# B&R Automation Studio project ui_test
Automation Studio 4.12.2.93; technology packages: mappView 5.19.0

## Configuration TS_UnitTest_Sample

CPU , AutomationRuntime F4.44, Build 6.3.0

### Task classes (Cpu.sw)
```
Cyclic#4 (cycle 10000 us, tolerance 10000000 us):
  SPL_CalcTe <- TS_UnitTest.Samples.Tests_Program.Tests_MyCalcLib_C.SPL_CalcTest.prg
  SPL_CalcT1 <- TS_UnitTest.Samples.Tests_Program.Tests_MyCalcLib_C.SPL_CalcTest_Variants.prg
  SPL_Assert <- TS_UnitTest.Samples.Framework_Extension_With_Custom_Asserts.SPL_AssertsEx.prg
  SPL_Asser1 <- TS_UnitTest.Samples.Framework_Features.SPL_Asserts.prg
  SPL_Behavi <- TS_UnitTest.Samples.Framework_Features.SPL_Behavior.prg
  utTemplate <- TS_UnitTest.Templates.HelperTool_Supported.utTemplate_automated.prg
  utTemplat1 <- TS_UnitTest.Templates.NoToolSupport.utTemplate_manual.prg
Binaries: iomap, asfw, arconfig, ashwd, sysconf
Libraries: Runtime, sys_lib, AsIecCon, astime, AsARCfg, AsBrStr, UnitTest, LibAssert1, UtWs, UtMgr, SPLMyCalc
```

### Hardware
```
PC_any : PC_any v1.1.0.0 (OrderNumber=PC)
  Cyclic1Duration = 100000
  Cyclic1Tolerance = 10000000
  Cyclic2Duration = 200000
  Cyclic2Tolerance = 10000000
  Cyclic3Duration = 500000
  Cyclic3Tolerance = 10000000
  Cyclic4Duration = 10000
  Cyclic4Tolerance = 10000000
  Cyclic5Duration = 2000000
  Cyclic5Tolerance = 10000000
  Cyclic6Duration = 3000000
  Cyclic6Tolerance = 12000000
  Cyclic7Duration = 4000000
  Cyclic7Tolerance = 12000000
  Cyclic8Duration = 5000000
  Cyclic8Tolerance = 30000000
```

## Configuration benchtop

CPU X20CP1381, AutomationRuntime G4.83, Build 4.1.2, Safety 0.0, Vc V4.72.6

### Task classes (Cpu.sw)
```
Cyclic#4:
  Program <- Program.prg
Libraries: AsBrStr, AsARCfg, runtime, sys_lib
```

### Hardware
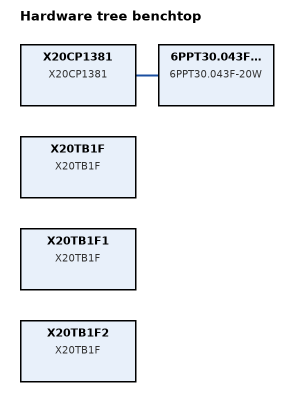
```
6PPT30.043F-20W : 6PPT30.043F-20W v1.3.5.0  [ETH1 -> X20CP1381.IF2 [Cable Type=PowerlinkCable, Length=10, Version=1.0.0.3]]
  Terminal = true
  PasswordVNC = 
  PasswordCIFS = 
  PasswordService = 
  VncKeyMappingFile = VC\6PPT30.043F-20W.dis
X20CP1381 : X20CP1381 v1.14.0.0  [X1 -> X1.SL; X2 -> X2.SL; X3 -> X3.SL]
  Module X1 (Type=X1, Virtual=true, Version=1.14.0.0)
    Connection (Connector=SS1, TargetModule=X20TB1F, TargetConnector=SS)
    Connection (Connector=SL, TargetModule=X20CP1381, TargetConnector=X1)
  Module X2 (Type=X2, Virtual=true, Version=1.14.0.0)
    Connection (Connector=SS1, TargetModule=X20TB1F1, TargetConnector=SS)
    Connection (Connector=SL, TargetModule=X20CP1381, TargetConnector=X2)
  Module X3 (Type=X3, Virtual=true, Version=1.14.0.0)
    Connection (Connector=SS1, TargetModule=X20TB1F2, TargetConnector=SS)
    Connection (Connector=SL, TargetModule=X20CP1381, TargetConnector=X3)
  Connector IF2:
    ActivateDevice = 1
  ConfigurationID = ui_test_benchtop
  ActivateOpcUa = 1
  OpcUaInformationModels_PV_Version = 1
X20TB1F : X20TB1F v1.0.0.0
X20TB1F1 : X20TB1F v1.0.0.0
X20TB1F2 : X20TB1F v1.0.0.0
```

## Logical view

Binary libraries used (declarations not repeated): operator, runtime, astime, AsIecCon, AsBrStr, AsARCfg, sys_lib, UnitTest, UtMgr, UtWs

### Global.var - Global variables
```iecst
VAR
	CurrentTemperature : INT;
	SetTemperature : INT;
END_VAR
```

### Package Logical/Libraries - Global libraries

- Visualisation Logical/mappView (not shown)

### Program Logical/Program (IEC)

#### Main.st
```iecst
PROGRAM _INIT
	SetTemperature := 35;
	CurrentTemperature;

END_PROGRAM

PROGRAM _CYCLIC

END_PROGRAM
```

### Package Logical/TS_UnitTest/Samples/Tests_Program - Unit test sample

### Library Logical/TS_UnitTest/Samples/Tests_Program/SPLMyCalc (IEC) - Simple Calculator
Depends on: Runtime

#### SPLMyCalc.typ - Exported data types
```iecst
(********************************************************************
 * COPYRIGHT -- Bernecker + Rainer
 ********************************************************************
 * Library: SPLMyCalc
 * File: SPLMyCalc.typ
 * Author: B+R
 ********************************************************************
 * Data types of library SPLMyCalc
 ********************************************************************)

TYPE
	MyCalcOperator_enum :
		( (*Enumerator of maths operations*)
		splMyCalcOPERATOR_RESET_OUTPUTS := 0, (*Resets the outputs. No calculation*)
		splMyCalcOPERATOR_ADD := 1, (*Add *)
		splMyCalcOPERATOR_SUBTRACT := 2, (*Subtract*)
		splMyCalcOPERATOR_MULTIPLICATION := 3, (*Multiplication*)
		splMyCalcOPERATOR_DIVISION := 4, (*Division*)
		splMyCalcOPERATOR_SQUARE := 5, (*Square of Param 1*)
		splMyCalcOPERATOR_EXP := 6 (*Param1 ^ Param2*)
		);
END_TYPE
```

#### SPLMyCalc.var - Exported constants
```iecst
(********************************************************************
 * COPYRIGHT --  Bernecker + Rainer
 ********************************************************************
 * Library: SPLMyCalc
 * File: SPLMyCalc.var
 * Author: B+R
 ********************************************************************
 * Constants of library SPLMyCalc
 ********************************************************************)
VAR CONSTANT
	splMyCalcERR_OUT_OF_RANGE : UINT := 50002;
	splMyCalcERR_NO_VALID_PARAM : UINT := 50001;
END_VAR
```

#### SPLMyCalc.fun - Exported functions and function blocks
```iecst
(********************************************************************
 * COPYRIGHT -- Bernecker + Rainer
 ********************************************************************
 * Library: SPLMyCalc
 * File: MyCalc.fun
 * Author: B+R
 ********************************************************************
 * Functions and function blocks of library SPLMyCalc
 ********************************************************************)

FUNCTION_BLOCK MyCalculator (*This functionblock provides several operations. If result is bigger / smaller than MIN or MAX, MIN or MAX are returned.*)
	VAR_INPUT
		CalcOperator : MyCalcOperator_enum; (*Calculation operation*)
		Param1 : INT; (*Paramerter 1*)
		Param2 : INT; (*Paramerter 2*)
	END_VAR
	VAR_OUTPUT
		Status : UINT; (*execution status: ERR_OK, ... *)
		Result : DINT; (*Result of the operation*)
	END_VAR
END_FUNCTION_BLOCK
```

#### SPLMyCalc.st
```iecst
(********************************************************************
 * COPYRIGHT -- Bernecker + Rainer
 ********************************************************************
 * Library: SPLMyCalc
 * File: SPLMyCalc.st
 * Author: B+R
 ********************************************************************
 * Implementation of library SPLMyCalc
 ********************************************************************)

(* This can be used as a sample for  Test Driven Development (TDD)/ Test First Development
Steps (in a nutshell):
    o Define your API (FB, functions, ...)
		 this is already done for the FB MyCalc
	o Create a new test program (by using the template)
	o Write a test case (e.g. Addition) for this FB.
		The tests should describe the expected behavior.
	o Transfer the test program to the target and run the test in the test view
		The test case will fail
	o Implement this FB (Addition), build and transfer, then run the test again
		The test case will pass
	o Write next test (e.g. Subtraction).
	..
	o Write test for MIN / MAX (underflow/overflow)
   	o Run the tests to verify your implementation.

Note:
	The sample test program in SPL_MyCalcLib_C provides some test cases using this FB.

 *)
FUNCTION_BLOCK MyCalculator

	Status := ERR_NOTIMPLEMENTED;

END_FUNCTION_BLOCK
```

### Package Logical/TS_UnitTest/Samples/Tests_Program/Tests_MyCalcLib_C - Tests SPLMyCalc with library "UnitTest"

### Program Logical/TS_UnitTest/Samples/Tests_Program/Tests_MyCalcLib_C/SPL_CalcTest (ANSIC) - Tests SPLMyCalc with library "UnitTest"

#### variables.var - PVs for the program and test suite
```iecst
(********************************************************************
 * COPYRIGHT -- Bernecker + Rainer
 ********************************************************************
 * Program: SPL_CalcTest
 * Author: B+R
 ********************************************************************
 * Local variables of program SPL_CalcTest
 * General variables - do not change
 ********************************************************************)
(*Describe the test*)
VAR
	Testsuite : UtMgrTestSuite := (Name:='SPL_MyCalcTests',Description:='Tests for MyCalc',Type:=utMgrTEST_TYPE_C,MetaInformation:='Some Meta Information can be added here');
END_VAR
(*Variables used in the tests*)
VAR
	instMyCalc : MyCalculator := (0);
END_VAR
```

#### testSuite.c - Handling of program and test suite
```c
/********************************************************************
 * COPYRIGHT -- Bernecker + Rainer
 ********************************************************************
 * Program: SPL_CalcTest
 * Author: B+R
 ********************************************************************
 * Test registration and handshake
 ********************************************************************/

#include <bur/plctypes.h>

#ifdef _DEFAULT_INCLUDES
#include <AsDefault.h>
#endif

#include "UnitTest.h"

void _INIT initTestSuite(void)
{
	utInit(&Testsuite);
}

void _CYCLIC cyclicWithTest(void)
{
	utCyclic(&Testsuite);
}

void _EXIT exitTestSuite(void)
{
	utExit(&Testsuite);
}
```

#### autoGeneratedFile.c - Auto generated code
```c
/*
B+R UnitTest: This is generated code.
Do not edit! Do not move!
Description: UnitTest Testprogramm infrastructure (List of TestSets).
LastUpdated: 2015-04-14 12:04:18Z
By B+R UnitTest Helper Version: 2.0.0.0
*/
#include "UnitTest.h"

UNITTEST_TESTSET_DECLARATION  testSet_MyCalcLib_Addition;
UNITTEST_TESTSET_DECLARATION  testSet_MyCalcLib_Subtraction;
UNITTEST_TESTSET_DECLARATION  testSet_MyCalcLib_Mult_Div;

UNITTEST_TESTSET_FIXTURES(utTestSets)
{
	new_TestSet(testSet_MyCalcLib_Addition),
	new_TestSet(testSet_MyCalcLib_Subtraction),
	new_TestSet(testSet_MyCalcLib_Mult_Div),
};
UNTITTEST_TESTSET_HANDLER();
```

#### testSet_MyCalcLib_Addition.c - Groups test cases for addition
```c
/********************************************************************
 * COPYRIGHT -- Bernecker + Rainer
 ********************************************************************
 * Program: SPL_CalcTest
 * Author: B+R
 ********************************************************************
 * Test set implementation
 ********************************************************************/

#include <bur/plctypes.h>

#ifdef _DEFAULT_INCLUDES
#include <AsDefault.h>
#endif

#include "UnitTest.h"

_TEST test_Add(void)
{
	/* initialize functionblock parameters */
	instMyCalc.CalcOperator = splMyCalcOPERATOR_ADD;
	instMyCalc.Param1   = 1;
	instMyCalc.Param2   = 2;
	/* call synchron functionblock */
	MyCalculator(&instMyCalc);

	/* check result */
	TEST_ASSERT_EQUAL_INT(3, instMyCalc.Result);
	TEST_ASSERT_EQUAL_INT(ERR_OK, instMyCalc.Status);

	/* test is done */
	TEST_DONE;
}

_TEST testResetOutputParam(void)
{

	/* Do any calculation with a result != 0  */
	instMyCalc.CalcOperator = splMyCalcOPERATOR_ADD;
	instMyCalc.Param1   = 1;
	instMyCalc.Param2   = 2;
	/* call synchron functionblock */
	MyCalculator(&instMyCalc);
	/* Please note: the result of the calculation isn't checked as this is not subject of this test case.	 */

	instMyCalc.CalcOperator = splMyCalcOPERATOR_RESET_OUTPUTS;
	/* call synchron functionblock */
	MyCalculator(&instMyCalc);

	/* check result */
	TEST_ASSERT_EQUAL_INT(0, instMyCalc.Result);
	TEST_ASSERT_EQUAL_INT(ERR_OK, instMyCalc.Status);

	/* test is done */
	TEST_DONE;

}

/* This test case shows an example of a test case that can be "false positive".
	As long as MyCalculator() is not implemented, this test passes.
	As long as instMyCalc.Result already is 0 when this test case will be called, it doesn't check wether the FB was called at all.
	--> There are several methods, to verify the FB was called and changed the variables that are used to prove functionality:
	Choose other parameter for an addition with negative values
	Before calling the FB set the output to any other value than the expected result. (e.g. By using _SETUP_TEST() and / or _TEARDOWN_TEST() )
	...

*/
_TEST test_Addition_negValue_badExampleParameter(void)
{
	/* initialize functionblock parameters */
	instMyCalc.CalcOperator = splMyCalcOPERATOR_ADD;
	instMyCalc.Param1   = -1;
	instMyCalc.Param2   = 1;
	/* call synchron functionblock */
	MyCalculator(&instMyCalc);

	/* check result */
	TEST_ASSERT_EQUAL_INT(0, instMyCalc.Result);
	TEST_ASSERT_EQUAL_INT(ERR_OK, instMyCalc.Status);

	/* test is done */
	TEST_DONE;
}

_TEST test_Addition_negValue(void)
{
	/* initialize functionblock parameters */
	instMyCalc.CalcOperator = splMyCalcOPERATOR_ADD;
	instMyCalc.Param1   = -1;
	instMyCalc.Param2   = 3;
	/* call synchron functionblock */
	MyCalculator(&instMyCalc);

	/* check result */
	TEST_ASSERT_EQUAL_INT(2, instMyCalc.Result);
	TEST_ASSERT_EQUAL_INT(ERR_OK, instMyCalc.Status);

	/* test is done */
	TEST_DONE;
}

/*
B+R UnitTest: This is generated code.
Do not edit! Do not move!
Description: UnitTest Testprogramm infrastructure (TestSet).
LastUpdated: 2015-04-14 12:04:18Z
By B+R UnitTest Helper Version: 2.0.0.0
*/
UNITTEST_FIXTURES(fixtures)
{
	new_TestFixture("test_Add", test_Add),
	new_TestFixture("testResetOutputParam", testResetOutputParam),
	new_TestFixture("test_Addition_negValue_badExampleParameter", test_Addition_negValue_badExampleParameter),
	new_TestFixture("test_Addition_negValue", test_Addition_negValue),
};

UNITTEST_CALLER_COMPLETE_EXPLICIT(testSet_MyCalcLib_Addition, "testSet_MyCalcLib_Addition", 0, 0, fixtures, 0, 0, 0);
```

#### testSet_MyCalcLib_Subtraction.c - Groups test cases for substraction
```c
/********************************************************************
 * COPYRIGHT -- Bernecker + Rainer
 ********************************************************************
 * Program: SPL_CalcTest
 * Author: B+R
 ********************************************************************
 * Test set implementation
 ********************************************************************/

#include <bur/plctypes.h>

#ifdef _DEFAULT_INCLUDES
#include <AsDefault.h>
#endif

#include "UnitTest.h"

_TEST test_Subtract(void)
{
	/* initialize functionblock parameters */
	instMyCalc.CalcOperator = splMyCalcOPERATOR_SUBTRACT;
	instMyCalc.Param1   = 4;
	instMyCalc.Param2   = 2;
	/* call synchron functionblock */
	MyCalculator(&instMyCalc);

	/* check result */
	TEST_ASSERT_EQUAL_INT(2, instMyCalc.Result);
	TEST_ASSERT_EQUAL_INT(ERR_OK, instMyCalc.Status);

	/* test is done */
	TEST_DONE;
}

_TEST test_Subtract_negResult(void)
{
	/* initialize functionblock parameters */
	instMyCalc.CalcOperator = splMyCalcOPERATOR_SUBTRACT;
	instMyCalc.Param1   = 6;
	instMyCalc.Param2   = 8;
	/* call synchron functionblock */
	MyCalculator(&instMyCalc);

	/* check result */
	TEST_ASSERT_EQUAL_INT(-2, instMyCalc.Result);
	TEST_ASSERT_EQUAL_INT(ERR_OK, instMyCalc.Status);

	/* test is done */
	TEST_DONE;
}

_TEST test_Subtract_zeroResult(void)
{
	/* initialize functionblock parameters */
	instMyCalc.CalcOperator = splMyCalcOPERATOR_SUBTRACT;
	instMyCalc.Param1   = 6;
	instMyCalc.Param2   = 6;
	/* call synchron functionblock */
	MyCalculator(&instMyCalc);

	/* check result */
	TEST_ASSERT_EQUAL_INT(0, instMyCalc.Result);
	TEST_ASSERT_EQUAL_INT(ERR_OK, instMyCalc.Status);

	/* test is done */
	TEST_DONE;
}

_TEST test_Subtract_boundaryArea_expect_MIN(void)
{
	/* initialize functionblock parameters */
	instMyCalc.CalcOperator = splMyCalcOPERATOR_SUBTRACT;
	instMyCalc.Param1   = -1;
	instMyCalc.Param2   = 32768;
	/* call synchron functionblock */
	MyCalculator(&instMyCalc);

	/* check result */
	TEST_ASSERT_EQUAL_INT(-32768, instMyCalc.Result);
	TEST_ASSERT_EQUAL_INT(splMyCalcERR_OUT_OF_RANGE, instMyCalc.Status);

	/* test is done */
	TEST_DONE;
}

/*
B+R UnitTest: This is generated code.
Do not edit! Do not move!
Description: UnitTest Testprogramm infrastructure (TestSet).
LastUpdated: 2015-04-14 12:04:18Z
By B+R UnitTest Helper Version: 2.0.0.0
*/
UNITTEST_FIXTURES(fixtures)
{
	new_TestFixture("test_Subtract", test_Subtract),
	new_TestFixture("test_Subtract_negResult", test_Subtract_negResult),
	new_TestFixture("test_Subtract_zeroResult", test_Subtract_zeroResult),
	new_TestFixture("test_Subtract_boundaryArea_expect_MIN", test_Subtract_boundaryArea_expect_MIN),
};

UNITTEST_CALLER_COMPLETE_EXPLICIT(testSet_MyCalcLib_Subtraction, "testSet_MyCalcLib_Subtraction", 0, 0, fixtures, 0, 0, 0);
```

#### testSet_MyCalcLib_Mult_Div.c - Groups test cases for multiplication and division
```c
/********************************************************************
 * COPYRIGHT -- Bernecker + Rainer
 ********************************************************************
 * Program: SPL_CalcTest
 * Author: B+R
 ********************************************************************
 * Test set implementation
 ********************************************************************/

#include <bur/plctypes.h>

#ifdef _DEFAULT_INCLUDES
#include <AsDefault.h>
#endif

#include "UnitTest.h"

_TEST test_Multiplication(void)
{
	/* initialize functionblock parameters */
	instMyCalc.CalcOperator = splMyCalcOPERATOR_MULTIPLICATION;
	instMyCalc.Param1   = 4;
	instMyCalc.Param2   = 4;
	/* call synchron functionblock */
	MyCalculator(&instMyCalc);
	/* check result */
	TEST_ASSERT_EQUAL_INT(16, instMyCalc.Result);
	TEST_ASSERT_EQUAL_INT(ERR_OK, instMyCalc.Status);
	/* test is done */
	TEST_DONE;
}

_TEST test_Division(void)
{
	/* initialize functionblock parameters */
	instMyCalc.CalcOperator = splMyCalcOPERATOR_DIVISION;
	instMyCalc.Param1   = 4;
	instMyCalc.Param2   = 4;
	/* call synchron functionblock */
	MyCalculator(&instMyCalc);

	/* check result */
	TEST_ASSERT_EQUAL_INT(1, instMyCalc.Result);
	TEST_ASSERT_EQUAL_INT(ERR_OK, instMyCalc.Status);

	/* test is done */
	TEST_DONE;
}

/*
B+R UnitTest: This is generated code.
Do not edit! Do not move!
Description: UnitTest Testprogramm infrastructure (TestSet).
LastUpdated: 2015-04-14 12:04:18Z
By B+R UnitTest Helper Version: 2.0.0.0
*/
UNITTEST_FIXTURES(fixtures)
{
	new_TestFixture("test_Multiplication", test_Multiplication),
	new_TestFixture("test_Division", test_Division),
};

UNITTEST_CALLER_COMPLETE_EXPLICIT(testSet_MyCalcLib_Mult_Div, "testSet_MyCalcLib_Mult_Div", 0, 0, fixtures, 0, 0, 0);
```

### Program Logical/TS_UnitTest/Samples/Tests_Program/Tests_MyCalcLib_C/SPL_CalcTest_Variants (ANSIC) - Examples how to avoid duplicated test code (advanced)

#### variables.var - PVs for the program and test suite
```iecst
(********************************************************************
 * COPYRIGHT -- Bernecker + Rainer
 ********************************************************************
 * Program: SPL_CalcTest_Variants
 * Author: B+R
 ********************************************************************
 * Local variables of program SPL_CalcTest_Variants
 * General variables - do not change
 ********************************************************************)
(*Describe the test*)
VAR
	Testsuite : UtMgrTestSuite := (Name:='SPL_CalcTest_Variants',Description:='Tests for MyCalc',Type:=utMgrTEST_TYPE_C,MetaInformation:='Some Meta Information can be added here');
END_VAR
(*Variables used in the tests*)
VAR
	instMyCalc : MyCalculator := (0);
END_VAR
```

#### testSuite.c - Handling of program and test suite
```c
/********************************************************************
 * COPYRIGHT -- Bernecker + Rainer
 ********************************************************************
 * Program: SPL_CalcTest_Variants
 * Author: B+R
 ********************************************************************
 * Test registration and handshake
 ********************************************************************/

#include <bur/plctypes.h>

#ifdef _DEFAULT_INCLUDES
#include <AsDefault.h>
#endif

#include "UnitTest.h"

void _INIT initTestSuite(void)
{
	utInit(&Testsuite);
}

void _CYCLIC cyclicWithTest(void)
{
	utCyclic(&Testsuite);
}

void _EXIT exitTestSuite(void)
{
	utExit(&Testsuite);
}
```

#### autoGeneratedFile.c - Auto generated code
```c
/*
B+R UnitTest: This is generated code.
Do not edit! Do not move!
Description: UnitTest Testprogramm infrastructure (List of TestSets).
LastUpdated: 2015-04-14 12:04:18Z
By B+R UnitTest Helper Version: 2.0.0.0
*/
#include "UnitTest.h"

UNITTEST_TESTSET_DECLARATION  testSet_MyCalcLib_Subtraction;
UNITTEST_TESTSET_DECLARATION  testSet_MyCalcLib_Subtraction_variantA;
UNITTEST_TESTSET_DECLARATION  testSet_MyCalcLib_Subtraction_variantB;
UNITTEST_TESTSET_DECLARATION  testSet_MyCalcLib_Subtraction_variantC;
UNITTEST_TESTSET_DECLARATION  testSet_MyCalcLib_Subtraction_variantD;

UNITTEST_TESTSET_FIXTURES(utTestSets)
{
	new_TestSet(testSet_MyCalcLib_Subtraction),
	new_TestSet(testSet_MyCalcLib_Subtraction_variantA),
	new_TestSet(testSet_MyCalcLib_Subtraction_variantB),
	new_TestSet(testSet_MyCalcLib_Subtraction_variantC),
	new_TestSet(testSet_MyCalcLib_Subtraction_variantD),
};
UNTITTEST_TESTSET_HANDLER();
```

#### testSet_MyCalcLib_Subtraction.c - Groups test cases for substraction
```c
/********************************************************************
 * COPYRIGHT -- Bernecker + Rainer
 ********************************************************************
 * Program: SPL_CalcTest_Variants
 * Author: B+R
 ********************************************************************
 * Test set implementation
 ********************************************************************/

#include <bur/plctypes.h>

#ifdef _DEFAULT_INCLUDES
#include <AsDefault.h>
#endif

#include "UnitTest.h"

_TEST test_Subtract(void)
{
	/* initialize functionblock parameters */
	instMyCalc.CalcOperator = splMyCalcOPERATOR_SUBTRACT;
	instMyCalc.Param1   = 4;
	instMyCalc.Param2   = 2;
	/* call synchron functionblock */
	MyCalculator(&instMyCalc);

	/* check result */
	TEST_ASSERT_EQUAL_INT(2, instMyCalc.Result);
	TEST_ASSERT_EQUAL_INT(ERR_OK, instMyCalc.Status);

	/* test is done */
	TEST_DONE;
}

_TEST test_Subtract_negResult(void)
{
	/* initialize functionblock parameters */
	instMyCalc.CalcOperator = splMyCalcOPERATOR_SUBTRACT;
	instMyCalc.Param1   = 6;
	instMyCalc.Param2   = 8;
	/* call synchron functionblock */
	MyCalculator(&instMyCalc);

	/* check result */
	TEST_ASSERT_EQUAL_INT(-2, instMyCalc.Result);
	TEST_ASSERT_EQUAL_INT(ERR_OK, instMyCalc.Status);

	/* test is done */
	TEST_DONE;
}

_TEST test_Subtract_zeroResult(void)
{
	/* initialize functionblock parameters */
	instMyCalc.CalcOperator = splMyCalcOPERATOR_SUBTRACT;
	instMyCalc.Param1   = 6;
	instMyCalc.Param2   = 6;
	/* call synchron functionblock */
	MyCalculator(&instMyCalc);

	/* check result */
	TEST_ASSERT_EQUAL_INT(0, instMyCalc.Result);
	TEST_ASSERT_EQUAL_INT(ERR_OK, instMyCalc.Status);

	/* test is done */
	TEST_DONE;
}

_TEST test_Subtract_boundaryArea_expect_MIN(void)
{
	/* initialize functionblock parameters */
	instMyCalc.CalcOperator = splMyCalcOPERATOR_SUBTRACT;
	instMyCalc.Param1   = -1;
	instMyCalc.Param2   = 32768;
	/* call synchron functionblock */
	MyCalculator(&instMyCalc);

	/* check result */
	TEST_ASSERT_EQUAL_INT(-32768, instMyCalc.Result);
	TEST_ASSERT_EQUAL_INT(splMyCalcERR_OUT_OF_RANGE, instMyCalc.Status);

	/* test is done */
	TEST_DONE;
}

/*
B+R UnitTest: This is generated code.
Do not edit! Do not move!
Description: UnitTest Testprogramm infrastructure (TestSet).
LastUpdated: 2015-04-14 12:04:18Z
By B+R UnitTest Helper Version: 2.0.0.0
*/
UNITTEST_FIXTURES(fixtures)
{
	new_TestFixture("test_Subtract", test_Subtract),
	new_TestFixture("test_Subtract_negResult", test_Subtract_negResult),
	new_TestFixture("test_Subtract_zeroResult", test_Subtract_zeroResult),
	new_TestFixture("test_Subtract_boundaryArea_expect_MIN", test_Subtract_boundaryArea_expect_MIN),
};

UNITTEST_CALLER_COMPLETE_EXPLICIT(testSet_MyCalcLib_Subtraction, "testSet_MyCalcLib_Subtraction", 0, 0, fixtures, 0, 0, 0);
```

#### testSet_MyCalcLib_Subtraction_variantA.c -  To check multiple subtraction combinations without code duplication a helper function can be created.
```c
/********************************************************************
 * COPYRIGHT -- Bernecker + Rainer
 ********************************************************************
 * Program: SPL_CalcTest_Variants
 * Author: B+R
 ********************************************************************
 * Test set implementation
 ********************************************************************/

#include <bur/plctypes.h>

#ifdef _DEFAULT_INCLUDES
#include <AsDefault.h>
#endif

#include "UnitTest.h"

/* To check multiple subtraction combinations without code duplication a helper function can be created.

Note: If an check (assert) is extracted into a helper function, the error report do not contain information about the parameters this helper function was called. For some use cases, this will be acceptable/OK for others not.
	See test_Subtract_MultipleCases()
One option to avoid this is to create multiple Test Cases each calling the same helper function once but with different parameters.
	See test_Subtract_1() and test_Subtract_boundaryArea_expect_MIN()  */
void verify_subtract(INT par1, INT par2 , DINT expectResult)
{
	instMyCalc.CalcOperator = splMyCalcOPERATOR_SUBTRACT;
	instMyCalc.Param1   = par1;
	instMyCalc.Param2   = par2;
	/* call synchron functionblock */
	MyCalculator(&instMyCalc);
	/* check result */
	TEST_ASSERT_EQUAL_INT(expectResult, instMyCalc.Result);
	TEST_ASSERT_EQUAL_INT(ERR_OK, instMyCalc.Status);
}

_TEST test_Subtract(void)
{
	verify_subtract(4, 2,2);

	/* test is done */
	TEST_DONE;
}

_TEST test_Subtract_negResult(void)
{
	verify_subtract(6, 8, -2);

	/* test is done */
	TEST_DONE;
}

_TEST test_Subtract_zeroResult(void)
{
	verify_subtract(6, 6, 0);

	/* test is done */
	TEST_DONE;
}

/* This test isn't reduced as there is (currently) no argument for  instMyCalc.Status  */
_TEST test_Subtract_boundaryArea_expect_MIN(void)
{
	/* initialize functionblock parameters */
	instMyCalc.CalcOperator = splMyCalcOPERATOR_SUBTRACT;
	instMyCalc.Param1   = -1;
	instMyCalc.Param2   = 32768;
	/* call synchron functionblock */
	MyCalculator(&instMyCalc);

	/* check result */
	TEST_ASSERT_EQUAL_INT(-32768, instMyCalc.Result);
	TEST_ASSERT_EQUAL_INT(splMyCalcERR_OUT_OF_RANGE, instMyCalc.Status);

	/* test is done */
	TEST_DONE;
}

/*
B+R UnitTest: This is generated code.
Do not edit! Do not move!
Description: UnitTest Testprogramm infrastructure (TestSet).
LastUpdated: 2015-04-14 12:04:18Z
By B+R UnitTest Helper Version: 2.0.0.0
*/
UNITTEST_FIXTURES(fixtures)
{
	new_TestFixture("test_Subtract", test_Subtract),
	new_TestFixture("test_Subtract_negResult", test_Subtract_negResult),
	new_TestFixture("test_Subtract_zeroResult", test_Subtract_zeroResult),
	new_TestFixture("test_Subtract_boundaryArea_expect_MIN", test_Subtract_boundaryArea_expect_MIN),
};

UNITTEST_CALLER_COMPLETE_EXPLICIT(testSet_MyCalcLib_Subtraction_variantA, "testSet_MyCalcLib_Subtraction_variantA", 0, 0, fixtures, 0, 0, 0);
```

#### testSet_MyCalcLib_Subtraction_variantB.c - TEST_ASSERT is used to output the parameters passed to the helper function when helper returns a failed.
```c
/********************************************************************
 * COPYRIGHT -- Bernecker + Rainer
 ********************************************************************
 * Program: SPL_CalcTest_Variants
 * Author: B+R
 ********************************************************************
 * Test set implementation
 ********************************************************************/

#include <bur/plctypes.h>

#ifdef _DEFAULT_INCLUDES
#include <AsDefault.h>
#endif

#include "UnitTest.h"

/* 	Create a helper returning a BOOL and pass the result of the helper to e.g. TEST_ASSERT()
Note: if the validation itself is not trivial, this function should be tested as well.

If the assert would be used in the helper as well, each of the checks count's twice.
Option would be, to use the TEST_INFO_LOC if returned false. */
BOOL verify_subtract_retBool(INT par1, INT par2 , DINT expectResult)
{
	instMyCalc.CalcOperator = splMyCalcOPERATOR_SUBTRACT;
	instMyCalc.Param1   = par1;
	instMyCalc.Param2   = par2;
	/* call synchron functionblock */
	MyCalculator(&instMyCalc);
	/* check result */
	return (expectResult == instMyCalc.Result);
}

_TEST test_Subtract(void)
{
	TEST_ASSERT(verify_subtract_retBool(4, 2, 2));

	/* test is done */
	TEST_DONE;
}

_TEST test_Subtract_negResult(void)
{
	TEST_ASSERT(verify_subtract_retBool(6, 8, -2));

	/* test is done */
	TEST_DONE;
}

_TEST test_Subtract_zeroResult(void)
{
	TEST_ASSERT(verify_subtract_retBool(6, 6, 0));

	/* test is done */
	TEST_DONE;
}

/* This test isn't reduced as there is (currently) no argument for  instMyCalc.Status  */
_TEST test_Subtract_boundaryArea_expect_MIN(void)
{
	/* initialize functionblock parameters */
	instMyCalc.CalcOperator = splMyCalcOPERATOR_SUBTRACT;
	instMyCalc.Param1   = -1;
	instMyCalc.Param2   = 32768;
	/* call synchron functionblock */
	MyCalculator(&instMyCalc);

	/* check result */
	TEST_ASSERT_EQUAL_INT(-32768, instMyCalc.Result);
	TEST_ASSERT_EQUAL_INT(splMyCalcERR_OUT_OF_RANGE, instMyCalc.Status);

	/* test is done */
	TEST_DONE;
}

/*
B+R UnitTest: This is generated code.
Do not edit! Do not move!
Description: UnitTest Testprogramm infrastructure (TestSet).
LastUpdated: 2015-04-14 12:04:18Z
By B+R UnitTest Helper Version: 2.0.0.0
*/
UNITTEST_FIXTURES(fixtures)
{
	new_TestFixture("test_Subtract", test_Subtract),
	new_TestFixture("test_Subtract_negResult", test_Subtract_negResult),
	new_TestFixture("test_Subtract_zeroResult", test_Subtract_zeroResult),
	new_TestFixture("test_Subtract_boundaryArea_expect_MIN", test_Subtract_boundaryArea_expect_MIN),
};

UNITTEST_CALLER_COMPLETE_EXPLICIT(testSet_MyCalcLib_Subtraction_variantB, "testSet_MyCalcLib_Subtraction_variantB", 0, 0, fixtures, 0, 0, 0);
```

#### testSet_MyCalcLib_Subtraction_variantC.c - When the helper is formulated as macro, the correct location (line / file) inside the testcase is given.
```c
/********************************************************************
 * COPYRIGHT -- Bernecker + Rainer
 ********************************************************************
 * Program: SPL_CalcTest_Variants
 * Author: B+R
 ********************************************************************
 * Test set implementation
 ********************************************************************/

#include <bur/plctypes.h>

#ifdef _DEFAULT_INCLUDES
#include <AsDefault.h>
#endif

#include "UnitTest.h"

#ifdef SMARTEDIT_DUMMY
/* When the helper is formulated as macro, the correct location (line / file) inside the testcase is given.
Each time the macro is used, the code gets duplicated.

Best practise: Extract a helper function first, use / test it before converting it into a macro, as functions can be far farbetter debugged / analyzed than macros. */
void def_verify_subtract(INT par1, INT par2 , DINT expectResult);
#endif
#define  def_verify_subtract( par1,  par2 , expectResult)\
{\
	instMyCalc.CalcOperator = splMyCalcOPERATOR_SUBTRACT;\
	instMyCalc.Param1   = par1;\
	instMyCalc.Param2   = par2;\
	/* call synchron functionblock */\
	MyCalculator(&instMyCalc);\
	/* check result */\
	TEST_ASSERT_EQUAL_INT(expectResult, instMyCalc.Result);\
	TEST_ASSERT_EQUAL_INT(ERR_OK, instMyCalc.Status);\
}

_TEST test_Subtract(void)
{
	def_verify_subtract(4, 2, 2);

	/* test is done */
	TEST_DONE;
}

_TEST test_Subtract_negResult(void)
{
	def_verify_subtract(6, 8, -2);
	/* test is done */
	TEST_DONE;
}

_TEST test_Subtract_zeroResult(void)
{
	def_verify_subtract(6, 6, 0);

	/* test is done */
	TEST_DONE;
}

/* This test isn't reduced as there is (currently) no argument for  instMyCalc.Status  */
_TEST test_Subtract_boundaryArea_expect_MIN(void)
{
	/* initialize functionblock parameters */
	instMyCalc.CalcOperator = splMyCalcOPERATOR_SUBTRACT;
	instMyCalc.Param1   = -1;
	instMyCalc.Param2   = 32768;
	/* call synchron functionblock */
	MyCalculator(&instMyCalc);

	/* check result */
	TEST_ASSERT_EQUAL_INT(-32768, instMyCalc.Result);
	TEST_ASSERT_EQUAL_INT(splMyCalcERR_OUT_OF_RANGE, instMyCalc.Status);

	/* test is done */
	TEST_DONE;
}

/*
B+R UnitTest: This is generated code.
Do not edit! Do not move!
Description: UnitTest Testprogramm infrastructure (TestSet).
LastUpdated: 2015-04-14 12:04:18Z
By B+R UnitTest Helper Version: 2.0.0.0
*/
UNITTEST_FIXTURES(fixtures)
{
	new_TestFixture("test_Subtract", test_Subtract),
	new_TestFixture("test_Subtract_negResult", test_Subtract_negResult),
	new_TestFixture("test_Subtract_zeroResult", test_Subtract_zeroResult),
	new_TestFixture("test_Subtract_boundaryArea_expect_MIN", test_Subtract_boundaryArea_expect_MIN),
};

UNITTEST_CALLER_COMPLETE_EXPLICIT(testSet_MyCalcLib_Subtraction_variantC, "testSet_MyCalcLib_Subtraction_variantC", 0, 0, fixtures, 0, 0, 0);
```

#### testSet_MyCalcLib_Subtraction_variantD.c - Custom Assert
```c
/********************************************************************
 * COPYRIGHT -- Bernecker + Rainer
 ********************************************************************
 * Program: SPL_CalcTest_Variants
 * Author: B+R
 ********************************************************************
 * Test set implementation
 ********************************************************************/

#include <bur/plctypes.h>

#ifdef _DEFAULT_INCLUDES
#include <AsDefault.h>
#endif

#include "UnitTest.h"

/*****************************************
* Begin Custom Assert

* Note: Custom asserts may be seperated from Test Sets.
* 		In this sample it's part of the Test Set file for symmetry reason
*
* Note: To learn more about Custom Asserts see help
*		or sample in \Logical\TS_UnitTest\Samples\Samples_Advanced_CustomAsserts\
 */
BOOL spl_verify_subtract_impl(INT par1, INT par2 , DINT expectResult,  unsigned long line, const char *file)
{
	instMyCalc.CalcOperator = splMyCalcOPERATOR_SUBTRACT;
	instMyCalc.Param1   = par1;
	instMyCalc.Param2   = par2;

	/* call synchron functionblock */
	MyCalculator(&instMyCalc);

	/* check expectations and report outcome */
	if(expectResult != instMyCalc.Result)
	{
		addFailure("Calculation Error", line, file);
	}
	else if (ERR_OK != instMyCalc.Status)
	{
		addFailure("Unexpected Status", line, file);
	}
	else
	{
		addPassed("",0,0);
		return 1;
	}
	return 0;
}

#ifdef SMARTEDIT_DUMMY
/* When the helper is formulated as macro, the correct location (line / file) inside the testcase is given. */
void SPL_ASSERT_VERIFY_SUBTRACT(INT par1, INT par2 , DINT expectResult);
#endif
#define  SPL_ASSERT_VERIFY_SUBTRACT( par1,  par2 , expectResult)  spl_verify_subtract_impl(par1, par2, expectResult, __LINE__, __FILE__);

/*****************************************
* End Custom Assert
*/

/*****************************************
	Begin Test Set
*/
_TEST test_Subtract(void)
{
	SPL_ASSERT_VERIFY_SUBTRACT(4, 2, 2);

	/* test is done */
	TEST_DONE;
}

_TEST test_Subtract_negResult(void)
{
	SPL_ASSERT_VERIFY_SUBTRACT(6, 8, -2);
	/* test is done */
	TEST_DONE;
}

_TEST test_Subtract_zeroResult(void)
{
	SPL_ASSERT_VERIFY_SUBTRACT(6, 6, 0);

	/* test is done */
	TEST_DONE;
}

/* This test isn't reduced as there is (currently) no argument for  instMyCalc.Status  */
_TEST test_Subtract_boundaryArea_expect_MIN(void)
{
	/* initialize functionblock parameters */
	instMyCalc.CalcOperator = splMyCalcOPERATOR_SUBTRACT;
	instMyCalc.Param1   = -1;
	instMyCalc.Param2   = 32768;
	/* call synchron functionblock */
	MyCalculator(&instMyCalc);

	/* check result */
	TEST_ASSERT_EQUAL_INT(-32768, instMyCalc.Result);
	TEST_ASSERT_EQUAL_INT(splMyCalcERR_OUT_OF_RANGE, instMyCalc.Status);

	/* test is done */
	TEST_DONE;
}

/*
B+R UnitTest: This is generated code.
Do not edit! Do not move!
Description: UnitTest Testprogramm infrastructure (TestSet).
LastUpdated: 2015-04-14 12:04:18Z
By B+R UnitTest Helper Version: 2.0.0.0
*/
UNITTEST_FIXTURES(fixtures)
{
	new_TestFixture("test_Subtract", test_Subtract),
	new_TestFixture("test_Subtract_negResult", test_Subtract_negResult),
	new_TestFixture("test_Subtract_zeroResult", test_Subtract_zeroResult),
	new_TestFixture("test_Subtract_boundaryArea_expect_MIN", test_Subtract_boundaryArea_expect_MIN),
};

UNITTEST_CALLER_COMPLETE_EXPLICIT(testSet_MyCalcLib_Subtraction_variantD, "testSet_MyCalcLib_Subtraction_variantD", 0, 0, fixtures, 0, 0, 0);
```

### Package Logical/TS_UnitTest/Samples/Framework_Extension_With_Custom_Asserts - Custom asserts

- Library Logical/TS_UnitTest/Samples/Framework_Extension_With_Custom_Asserts/LibAssert1 (ANSIC) - Sample library: Creation of custom asserts (no source held here)

### Program Logical/TS_UnitTest/Samples/Framework_Extension_With_Custom_Asserts/SPL_AssertsEx (ANSIC) - This sample uses custom asserts defined in LibAssert1

#### README.txt
```
Please note

The samples in this program provides no good programming style!
They are solely for demonstrating the behavior of the framework.
Bad style:
	o	There is no test of any function or FB, just asserts failing or passing (depending on PV values)
	o	Expectations are variables and no constants
	o	Results are constants instead of results / outputs
	o	Mulitple asserts per Test Case
```

#### testSuite.var
```iecst
(********************************************************************
 * COPYRIGHT -- Bernecker + Rainer
 ********************************************************************
 * Program: SPL_AssertsEx
 * Author: B+R
 ********************************************************************
 * Local variables of program SPL_AssertsEx
 * General variables
 ********************************************************************)
VAR
	Testsuite : UtMgrTestSuite := (Name:='SPL_CustomAsserts',Description:='The sample custom asserts are defined in LibAssert1. This test shows their usage.',Type:=utMgrTEST_TYPE_C);
END_VAR
```

#### testSuite.c
```c
/********************************************************************
 * COPYRIGHT -- Bernecker + Rainer
 ********************************************************************
 * Program: SPL_AssertsEx
 * Author: B+R
 ********************************************************************
 * Test registration and handshake
 ********************************************************************/

#include <bur/plctypes.h>

#ifdef _DEFAULT_INCLUDES
#include <AsDefault.h>
#endif

#include "UnitTest.h"

void _INIT initTestSuite(void)
{
	utInit(&Testsuite);
}

void _CYCLIC cyclicWithTest(void)
{
	/* Some code */
	utCyclic(&Testsuite);
}

void _EXIT exitTestSuite(void)
{
	utExit(&Testsuite);
}
```

#### autoGeneratedFile.c
```c
/*
B+R UnitTest: This is generated code.
Do not edit! Do not move!
Description: UnitTest Testprogramm infrastructure (List of TestSets).
LastUpdated: 2015-04-14 12:04:08Z
By B+R UnitTest Helper Version: 2.0.0.0
*/
#include "UnitTest.h"

UNITTEST_TESTSET_DECLARATION  testSet_AssertsExt;

UNITTEST_TESTSET_FIXTURES(utTestSets)
{
	new_TestSet(testSet_AssertsExt),
};
UNTITTEST_TESTSET_HANDLER();
```

#### varAssertExt.var - Variables used in testSet_AssertsExt
```iecst
(********************************************************************
 * COPYRIGHT -- Bernecker + Rainer
 ********************************************************************
 * Program: SPL_AssertsEx
 * Author: B+R
 ********************************************************************
 * Local variables of program SPL_AssertsEx
 * For test set testSet_AssertsExt.c
 ********************************************************************)
VAR
	FloatArrayDeltaForComparison : ARRAY[0..50] OF REAL;
	FloatArray2 : ARRAY[0..50] OF REAL;
	FloatArray1 : ARRAY[0..50] OF REAL;
END_VAR
```

#### testSet_AssertsExt.c - Uses Assertions of Library utAssertExt
```c
/********************************************************************
* COPYRIGHT -- Bernecker + Rainer
********************************************************************
* Program: SPL_AssertsEx
* Author: B+R
********************************************************************
* This test set shows the use of self created asserts.
* Asserts are implemented in the library LibAssert1.
********************************************************************/

#include <bur/plctypes.h>

#ifdef _DEFAULT_INCLUDES
#include <AsDefault.h>
#endif

#include "UnitTest.h"
#include "LibAssert1.h"

_TEST test_splAssert_ArrayOfRealValues(void)
{
	/* manual generated differences for demonstration of the SPL_ASSERT */
	FloatArray1[0] = 2;
	FloatArray2[0] = 2;

	FloatArray1[1] = 3;
	FloatArray2[1] = 1;

	FloatArray1[30] = 3.33;
	FloatArray2[30] = 1.11;

	FloatArrayDeltaForComparison[31] = 1; /* Within -> pass, equal -> failed */
	FloatArray1[31] = 3.33;
	FloatArray2[31] = 3.31;

	SPL_ASSERT_ARRAY_EQUAL_REAL(FloatArray1, FloatArray2, sizeof(FloatArray1) / sizeof(FloatArray1[0]) );
	SPL_ASSERT_ARRAY_REAL_WITHIN(FloatArrayDeltaForComparison, FloatArray1, FloatArray2, sizeof(FloatArray1) / sizeof(FloatArray1[0]) );
	TEST_DONE;
}

_TEST test_splAssert_Boundary()
{
	/* should fail */
	SPL_ASSERT_UPPER_BOUNDARY(2,4);

	/* should pass */
	SPL_ASSERT_UPPER_BOUNDARY(4,2);

	TEST_DONE;
}

/*
B+R UnitTest: This is generated code.
Do not edit! Do not move!
Description: UnitTest Testprogramm infrastructure (TestSet).
LastUpdated: 2015-04-14 12:04:07Z
By B+R UnitTest Helper Version: 2.0.0.0
*/
UNITTEST_FIXTURES(fixtures)
{
	new_TestFixture("test_splAssert_ArrayOfRealValues", test_splAssert_ArrayOfRealValues),
	new_TestFixture("test_splAssert_Boundary", test_splAssert_Boundary),
};

UNITTEST_CALLER_COMPLETE_EXPLICIT(testSet_AssertsExt, "testSet_AssertsExt", 0, 0, fixtures, 0, 0, 0);
```

### Package Logical/TS_UnitTest/Samples/Framework_Features - Framework features

### Program Logical/TS_UnitTest/Samples/Framework_Features/SPL_Asserts (ANSIC) - Available basic asserts

#### README.txt
```
Please note

The samples in this program provides no good programming style!
They are solely for demonstrating the behavior of the framework.
Bad style:
	o	There is no test of any function or FB, just asserts failing or passing (depending on PV values)
	o	Expectations are variables and no constants
	o	Mulitple asserts per Test Case
```

#### testSuite.var
```iecst
(********************************************************************
 * COPYRIGHT -- Bernecker + Rainer
 ********************************************************************
 * Program: SPL_Asserts
 * Author: B+R
 ********************************************************************
 * Local variables of program SPL_Asserts
 * General variables
 ********************************************************************)
VAR
	Testsuite : UtMgrTestSuite := (Name:='SPL_Asserts',Description:='Shows asserts and usage',Type:=utMgrTEST_TYPE_C);
END_VAR
```

#### testSuite.c - Handling of program and test suite
```c
/********************************************************************
 * COPYRIGHT -- Bernecker + Rainer
 ********************************************************************
 * Program: SPL_Asserts
 * Author: B+R
 ********************************************************************
 * Test registration and handshake
 ********************************************************************/

#include <bur/plctypes.h>

#ifdef _DEFAULT_INCLUDES
#include <AsDefault.h>
#endif

#include "UnitTest.h"

void _INIT initTestSuite(void)
{
	utInit(&Testsuite);
}

void _CYCLIC cyclicWithTest(void)
{
	/* Some code */
	utCyclic(&Testsuite);
}

void _EXIT exitTestSuite(void)
{
	utExit(&Testsuite);
}
```

#### autoGeneratedFile.c - Auto generated code
```c
/*
B+R UnitTest: This is generated code.
Do not edit! Do not move!
Description: UnitTest Testprogramm infrastructure (List of TestSets).
LastUpdated: 2015-04-14 12:03:48Z
By B+R UnitTest Helper Version: 2.0.0.0
*/
#include "UnitTest.h"

UNITTEST_TESTSET_DECLARATION  testSet_Asserts;

UNITTEST_TESTSET_FIXTURES(utTestSets)
{
	new_TestSet(testSet_Asserts),
};
UNTITTEST_TESTSET_HANDLER();
```

#### varAsserts.var - Variables used in testSet_Asserts
```iecst
(********************************************************************
 * COPYRIGHT -- Bernecker + Rainer
 ********************************************************************
 * Program: SPL_Asserts
 * Author: B+R
 ********************************************************************
 * Local variables of program SPL_Asserts
 * For test set testSet_Asserts.c
 ********************************************************************)
VAR
	Buffer1 : ARRAY[0..9] OF USINT := [10(0)];
	Buffer2 : ARRAY[0..19] OF USINT := [20(0)];
	MySecondVar : UDINT := 2;
	Pointer : REFERENCE TO UDINT;
	ConditionFlag : BOOL := FALSE;
END_VAR
(*Strings*)
VAR
	String1 : STRING[80] := '';
	String2 : STRING[80] := '';
	WString1 : WSTRING[80] := "World";
	WString2 : WSTRING[80] := "Hello";
END_VAR
(*Integer*)
VAR
	Si1 : SINT := 0;
	Si2 : SINT := 0;
	Usi1 : USINT := 0;
	Usi2 : USINT := 0;
	I1 : INT := 0;
	I2 : INT := 0;
	Ui1 : UINT := 0;
	Ui2 : UINT := 0;
	Di1 : DINT := 0;
	Di2 : DINT := 0;
	Udi1 : UDINT := 0;
	Udi2 : UDINT := 0;
END_VAR
(*Floatingpoint*)
VAR
	LReal2 : REAL;
	LRealDeltaForComparison : REAL;
	LReal1 : REAL;
	Real2 : REAL;
	RealDeltaForComparison : REAL;
	Real1 : REAL;
END_VAR
```

#### testSet_Asserts.c - Available Asserts
```c
/********************************************************************
* COPYRIGHT -- Bernecker + Rainer
********************************************************************
* Program: SPL_Asserts
* Author: B+R
********************************************************************
* This test set shows the available asserts of the UnitTest library
********************************************************************/

#include <bur/plctypes.h>

#ifdef _DEFAULT_INCLUDES
#include <AsDefault.h>
#endif

#include "UnitTest.h"

/* Executed before each test case */
_SETUP_TEST(void)
{
	MySecondVar = 2;

	TEST_DONE;
}

/* Executed after each test case */
_TEARDOWN_TEST(void)
{
	TEST_DONE;
}

_TEST test_int(void)
{
	TEST_ASSERT_EQUAL_INT(	Usi1, 	Usi2);
	TEST_ASSERT_EQUAL_INT( 	Si1,	Si2 );
	TEST_ASSERT_EQUAL_INT( 	Ui1, 	Ui2	);
	TEST_ASSERT_EQUAL_INT( 	I1, 	I2	);
	TEST_ASSERT_EQUAL_INT( 	Di1, 	Di2	);
	TEST_ASSERT_EQUAL_INT(	Udi1, 	Udi2);

	TEST_DONE;
}

_TEST test_string(void)
{
	TEST_ASSERT_EQUAL_STRING(String1, String2 );

	TEST_DONE;
}

_TEST test_wstring(void)
{
	TEST_ASSERT_EQUAL_WSTRING(WString1,	WString2);

	TEST_DONE;
}

_TEST test_float(void)
{
	TEST_ASSERT_EQUAL_FLOAT(Real1, Real2);
	TEST_ASSERT_FLOAT_WITHIN(RealDeltaForComparison, Real1, Real2);

	TEST_ASSERT_EQUAL_REAL(Real1, Real2);
	TEST_ASSERT_REAL_WITHIN(RealDeltaForComparison, Real1, Real2);

	TEST_DONE;
}

_TEST test_double(void)
{
	TEST_ASSERT_EQUAL_DOUBLE(LReal1, LReal2);
	TEST_ASSERT_DOUBLE_WITHIN(LRealDeltaForComparison, LReal1, LReal2);

	TEST_ASSERT_EQUAL_LREAL(LReal1, LReal2);
	TEST_ASSERT_LREAL_WITHIN(LRealDeltaForComparison, LReal1, LReal2);

	TEST_DONE;
}

_TEST test_memory(void)
{
	TEST_ASSERT_EQUAL_MEM(Buffer1, Buffer2, sizeof(Buffer1)  );

	TEST_DONE;
}

_TEST test_null_true_and_false(void)
{
	TEST_ASSERT_NOT_NULL(Pointer);
	TEST_ASSERT_NOT_NULL(0); 	/* Not Ok */

	TEST_ASSERT_NULL(0); 		/* Ok */
	TEST_ASSERT_NULL(Pointer);

	Pointer = &Udi1;
	TEST_ASSERT_NULL(Pointer); /* Not Ok */

	TEST_DONE;
}

_TEST test_message(void)
{
	TEST_ASSERT_MESSAGE(ConditionFlag, "This text, if condition evaluates to false.");
	ConditionFlag = 0;
	TEST_ASSERT_MESSAGE(ConditionFlag, "This text, because condition evaluates to false.");
	ConditionFlag = 4;
	TEST_ASSERT_MESSAGE(ConditionFlag, "Nothing, as condition evaluates to true (!= 0).");

	TEST_DONE;
}

_TEST test_info(void)
{
	TEST_INFO("Info Text - for some comment");
	TEST_INFO_POS("Info Text - for some comment with position");

	TEST_DONE;
}

_TEST test_fail(void)
{
	TEST_FAIL("Always fails");

	TEST_DONE;
}

/*
B+R UnitTest: This is generated code.
Do not edit! Do not move!
Description: UnitTest Testprogramm infrastructure (TestSet).
LastUpdated: 2015-04-14 12:03:48Z
By B+R UnitTest Helper Version: 2.0.0.0
*/
UNITTEST_FIXTURES(fixtures)
{
	new_TestFixture("test_int", test_int),
	new_TestFixture("test_string", test_string),
	new_TestFixture("test_wstring", test_wstring),
	new_TestFixture("test_float", test_float),
	new_TestFixture("test_double", test_double),
	new_TestFixture("test_memory", test_memory),
	new_TestFixture("test_null_true_and_false", test_null_true_and_false),
	new_TestFixture("test_message", test_message),
	new_TestFixture("test_info", test_info),
	new_TestFixture("test_fail", test_fail),
};

UNITTEST_CALLER_COMPLETE_EXPLICIT(testSet_Asserts, "testSet_Asserts", setupTest, teardownTest, fixtures, 0, 0, 0);
```

### Program Logical/TS_UnitTest/Samples/Framework_Features/SPL_Behavior (ANSIC) - This sample is about the control flow of test programs

#### README.txt
```
Please note

The samples in this program provides no good programming style!
They are solely for demonstrating the behavior of the framework.
Bad style:
	o	Asserts should only be used to verify the test case as the report should be short ans meaningful (No explainings, just the relevant facts).
	o	Asserts should only be used in test cases.
	o	Test cases should be named meaningful.
	o	Macros are used instead of helper functions.
```

#### testSuite.var
```iecst
(********************************************************************
 * COPYRIGHT -- Bernecker + Rainer
 ********************************************************************
 * Program: SPL_Behavior
 * Author: B+R
 ********************************************************************
 * Local variables of program SPL_Behavior
 * General variables
 ********************************************************************)
VAR
	Testsuite : UtMgrTestSuite := (Name:='SPL_framework_behavior',Description:='Every TestSet provides an independend sample to show the behavior of a set',Type:=utMgrTEST_TYPE_C);
END_VAR
```

#### testSuite.c - Handling of program and test suite
```c
/********************************************************************
 * COPYRIGHT -- Bernecker + Rainer
 ********************************************************************
 * Program: SPL_Behavior
 * Author: B+R
 ********************************************************************
 * Test registration and handshake
 ********************************************************************/

#include <bur/plctypes.h>

#ifdef _DEFAULT_INCLUDES
#include <AsDefault.h>
#endif

#include "UnitTest.h"

#include "iPrototypes.h"

void _INIT initTestSuite(void)
{
	utInit(&Testsuite);
}

void _CYCLIC cyclicWithTest(void)
{
	/* Some code */
	utCyclic(&Testsuite);

	if(Testsuite.TestFinishedDone)
	{
		resetDataForTestSet_Complete();
		resetDataForTestSet_TestCases();
		resetDataForTestSet_SetSetupTeardown();
		resetDataForTestSet_TestSetupTeardown();
	}
}

void _EXIT exitTestSuite(void)
{
	utExit(&Testsuite);
}
```

#### autoGeneratedFile.c - Auto generated code
```c
/*
B+R UnitTest: This is generated code.
Do not edit! Do not move!
Description: UnitTest Testprogramm infrastructure (List of TestSets).
LastUpdated: 2015-04-14 12:03:48Z
By B+R UnitTest Helper Version: 2.0.0.0
*/
#include "UnitTest.h"

UNITTEST_TESTSET_DECLARATION  test_SetTestCases;
UNITTEST_TESTSET_DECLARATION  test_SetTestCases_SetSetup_SetTeardown;
UNITTEST_TESTSET_DECLARATION  test_SetTestCases_TestSetup_TestTeardown;
UNITTEST_TESTSET_DECLARATION  test_SetComplete;
UNITTEST_TESTSET_DECLARATION  TestBusy_Asyncronous;
UNITTEST_TESTSET_DECLARATION  TestBusy_Asyncronous_with_CyclicSet;

UNITTEST_TESTSET_FIXTURES(utTestSets)
{
	new_TestSet(test_SetTestCases),
	new_TestSet(test_SetTestCases_SetSetup_SetTeardown),
	new_TestSet(test_SetTestCases_TestSetup_TestTeardown),
	new_TestSet(test_SetComplete),
	new_TestSet(TestBusy_Asyncronous),
	new_TestSet(TestBusy_Asyncronous_with_CyclicSet),
};
UNTITTEST_TESTSET_HANDLER();
```

#### iPrototypes.h
```c
/********************************************************************
 * COPYRIGHT -- Bernecker + Rainer
 ********************************************************************
 * Program: SPL_Behavior
 * File: iPrototypes.h
 * Author: B+R
 *******************************************************************/

#include <bur/plctypes.h>

/* Prototyping of functions  */
void 	resetDataForTestSet();
void 	checkAndWriteCounterIfChanged( unsigned long line, const char *file);

void	resetDataForTestSet_Complete();
void	resetDataForTestSet_TestCases();
void	resetDataForTestSet_SetSetupTeardown();
void	resetDataForTestSet_TestSetupTeardown();
```

#### iHelperFunction.h
```c
/********************************************************************
 * COPYRIGHT -- Bernecker + Rainer
 ********************************************************************
 * Program: SPL_Behavior
 * File: iHelperFunction.h
 * Author: B+R
 *******************************************************************/

#include <bur/plctypes.h>

#include "iPrototypes.h"

/* This Macro is for tracing the calls in the sample
(For exemplification)*/
#define LOG_FOR_EXEMPLIFICATION_CYCLIC_SET  \
	brsstrcat((UDINT)OutputString, (UDINT)"Cyclic set - "); \
	checkAndWriteCounterIfChanged(__LINE__, __FILE__); \
	CounterInSet++;

/* This Macro is for tracing the calls in the sample
(For exemplification)*/
#define LOG_FOR_EXEMPLIFICATION_TEST_CASE_1   \
	brsstrcat((UDINT)OutputString,(UDINT) "Call test 1 - "); \
	checkAndWriteCounterIfChanged(__LINE__, __FILE__);

/* This Macro is for tracing the calls in the sample
(For exemplification)*/
#define LOG_FOR_EXEMPLIFICATION_TEST_CASE_2 \
	brsstrcat((UDINT)OutputString,(UDINT) "Call test 2 - "); \
	checkAndWriteCounterIfChanged(__LINE__, __FILE__);

/* This Macro is for tracing the calls in the sample
(For exemplification)*/
#define LOG_FOR_EXEMPLIFICATION_TEST_CASE_3   \
	brsstrcat((UDINT)OutputString,(UDINT) "Call test 3 - "); \
	checkAndWriteCounterIfChanged(__LINE__, __FILE__);

/* This Macro is for tracing the calls in the sample
(For exemplification)*/
#define LOG_FOR_EXEMPLIFICATION_SETUP_SET  \
	brsstrcat((UDINT)OutputString, (UDINT)"Setup set - "); \
	checkAndWriteCounterIfChanged(__LINE__, __FILE__);

/* This Macro is for tracing the calls in the sample
(For exemplification)*/
#define LOG_FOR_EXEMPLIFICATION_TEARDOWN_SET  \
	brsstrcat((UDINT)OutputString, (UDINT)"Teardown set - "); \
	checkAndWriteCounterIfChanged(__LINE__, __FILE__);

 /* This Macro is for tracing the calls in the sample
(For exemplification)*/
#define LOG_FOR_EXEMPLIFICATION_SETUP_TEST \
	brsstrcat((UDINT)OutputString, (UDINT)"Setup test - "); \
	checkAndWriteCounterIfChanged(__LINE__, __FILE__);

/* This Macro is for tracing the calls in the sample
(For exemplification)*/
#define LOG_FOR_EXEMPLIFICATION_TEARDOWN_TEST  \
	brsstrcat((UDINT)OutputString, (UDINT)"Teardown test - "); \
	checkAndWriteCounterIfChanged(__LINE__, __FILE__);

/* ************************************************/

/* Add this line behind a LOG_FOR_EXEMPLIFICATION_TEST_CASE_x to simulate an asyncron test case
 This Macro is for tracing the calls in the sample
(For exemplification)*/
#define LOG_FOR_EXEMPLIFICATION_TEST_BUSY  if(CountTestCaseRuns < DEF_BUSY_STEPS)\
	{\
	countTestCaseRuns++; \
	brsstrcat((UDINT)OutputString,(UDINT) "TEST_BUSY (recall in next cycle) - "); \
	TEST_BUSY; } \
	else { CountTestCaseRuns = 0;}
```

#### iHelperFunction.c
```c
/********************************************************************
 * COPYRIGHT -- Bernecker + Rainer
 ********************************************************************
 * Program: SPL_Behavior
 * File: iHelperFunction.c
 * Author: B+R
 *******************************************************************/

#include <bur/plctypes.h>

#ifdef _DEFAULT_INCLUDES
#include <AsDefault.h>
#endif

#include "UnitTest.h"
#include "AsBrStr.h"
#include "iPrototypes.h"

void resetDataForTestSet()
{
	brsstrcpy((UDINT)OutputString, (UDINT)"");
	CounterInSet = 0;
	CounterInSet_LastChecked = -1;
	CounterToStringBuffer[0] = 0;
}

void checkAndWriteCounterIfChanged( unsigned long line, const char *file)
{
	if(CounterInSet_LastChecked != CounterInSet)
	{
		addFailure((char*)OutputString, line, file);

		CounterInSet_LastChecked = CounterInSet;
		brsitoa(CounterInSet + 1, (UDINT) CounterToStringBuffer);

		brsstrcpy((UDINT)OutputString, (UDINT)"( ");
		brsstrcat((UDINT)OutputString, (UDINT)CounterToStringBuffer);
		/*		brsstrcat((UDINT)OutputString, (UDINT)". task cylce in TestSet) "); */
		brsstrcat((UDINT)OutputString, (UDINT)". cylce) ");

		addFailure((char*)OutputString, line, file);

	}
	else if(OutputString[0])
	{
		/*		TEST_FAIL(OutputString);*/
		addFailure((char*)OutputString, line, file);
	}

}
```

#### controlFlowVariables.var - Variables used in sub package "ControlFlow"
```iecst
(********************************************************************
 * COPYRIGHT -- Bernecker + Rainer
 ********************************************************************
 * Program: SPL_Behavior
 * File: controlFlowVariables.var
 * Author: B+R
 ********************************************************************
 * Local variables of program SPL_Behavior
 ********************************************************************)
VAR
	CounterInSet : DINT := 0;
	CounterInSet_LastChecked : DINT := 0;
	OutputString : STRING[200];
	CounterToStringBuffer : STRING[20] := '';
END_VAR
(*Warning "Warning : 'CountTestCaseRuns' defined but not used" can be ignored.
Warnings for this variable occurs when no LOG_FOR_EXEMPLIFICATION_TEST_BUSY is used inside a set. *)
VAR CONSTANT
	DEF_BUSY_STEPS : USINT := 2;
END_VAR
VAR
	CountTestCaseRuns : USINT := 0;
END_VAR
```

#### Package Logical/TS_UnitTest/Samples/Framework_Features/SPL_Behavior/ControlFlow - Shows sequence of calls within test set (depending on the defined optional handles)

#### test_SetTestCases.c
```c
/********************************************************************
* COPYRIGHT -- Bernecker + Rainer
********************************************************************
* Program: SPL_Behavior
* Author: B+R
********************************************************************
* This test set shows the sequence of calls within a test set
* Add some busy conditions or test cases to see the changes.
********************************************************************/

#include <bur/plctypes.h>

#ifdef _DEFAULT_INCLUDES
#include <AsDefault.h>
#endif

#include "UnitTest.h"

#include "iHelperFunction.h"

void resetDataForTestSet_TestCases()
{
	resetDataForTestSet();
}

_CYCLIC_SET(void)
{
	LOG_FOR_EXEMPLIFICATION_CYCLIC_SET;

	return;
}

_TEST test_1(void)
{
	LOG_FOR_EXEMPLIFICATION_TEST_CASE_1;

	TEST_DONE;
}

_TEST test_2(void)
{
	LOG_FOR_EXEMPLIFICATION_TEST_CASE_2;

	TEST_DONE;
}

_TEST test_3(void)
{
	LOG_FOR_EXEMPLIFICATION_TEST_CASE_3;

	TEST_DONE;
}

/*
B+R UnitTest: This is generated code.
Do not edit! Do not move!
Description: UnitTest Testprogramm infrastructure (TestSet).
LastUpdated: 2015-04-14 12:03:48Z
By B+R UnitTest Helper Version: 2.0.0.0
*/
UNITTEST_FIXTURES(fixtures)
{
	new_TestFixture("test_1", test_1),
	new_TestFixture("test_2", test_2),
	new_TestFixture("test_3", test_3),
};

UNITTEST_CALLER_COMPLETE_EXPLICIT(test_SetTestCases, "test_SetTestCases", 0, 0, fixtures, 0, 0, cyclicSetCaller);
```

#### test_SetTestCases_SetSetup_SetTeardown.c
```c
/********************************************************************
* COPYRIGHT -- Bernecker + Rainer
********************************************************************
* Program: SPL_Behavior
* Author: B+R
********************************************************************
* This test set shows the sequence of calls within a test set
* Add some busy conditions or test cases to see the changes.
********************************************************************/

#include <bur/plctypes.h>

#ifdef _DEFAULT_INCLUDES
#include <AsDefault.h>
#endif

#include "UnitTest.h"

#include "iHelperFunction.h"

void resetDataForTestSet_SetSetupTeardown()
{
	resetDataForTestSet();
}

_CYCLIC_SET(void)
{
	LOG_FOR_EXEMPLIFICATION_CYCLIC_SET;
	return;
}

_SETUP_SET(void)
{
	LOG_FOR_EXEMPLIFICATION_SETUP_SET;
	TEST_DONE;
}

_TEARDOWN_SET(void)
{
	LOG_FOR_EXEMPLIFICATION_TEARDOWN_SET;
	TEST_DONE;
}

_TEST test_1(void)
{
	LOG_FOR_EXEMPLIFICATION_TEST_CASE_1;
	TEST_DONE;
}

_TEST test_2(void)
{
	LOG_FOR_EXEMPLIFICATION_TEST_CASE_2;
	TEST_DONE;
}

_TEST test_3(void)
{
	LOG_FOR_EXEMPLIFICATION_TEST_CASE_3;
	TEST_DONE;
}

/*
B+R UnitTest: This is generated code.
Do not edit! Do not move!
Description: UnitTest Testprogramm infrastructure (TestSet).
LastUpdated: 2015-04-14 12:03:48Z
By B+R UnitTest Helper Version: 2.0.0.0
*/
UNITTEST_FIXTURES(fixtures)
{
	new_TestFixture("test_1", test_1),
	new_TestFixture("test_2", test_2),
	new_TestFixture("test_3", test_3),
};

UNITTEST_CALLER_COMPLETE_EXPLICIT(test_SetTestCases_SetSetup_SetTeardown, "test_SetTestCases_SetSetup_SetTeardown", 0, 0, fixtures, setupSet, teardownSet, cyclicSetCaller);
```

#### test_SetTestCases_TestSetup_TestTeardown.c
```c
/********************************************************************
* COPYRIGHT -- Bernecker + Rainer
********************************************************************
* Program: SPL_Behavior
* Author: B+R
********************************************************************
* This test set shows the sequence of calls within a test set
* Add some busy conditions or test cases to see the changes.
********************************************************************/

#include <bur/plctypes.h>

#ifdef _DEFAULT_INCLUDES
#include <AsDefault.h>
#endif

#include "UnitTest.h"

#include "iHelperFunction.h"

void resetDataForTestSet_TestSetupTeardown()
{
	resetDataForTestSet();
}

_CYCLIC_SET(void)
{
	LOG_FOR_EXEMPLIFICATION_CYCLIC_SET;
	return;
}

_SETUP_TEST(void)
{
	LOG_FOR_EXEMPLIFICATION_SETUP_TEST;
	TEST_DONE;
}

_TEARDOWN_TEST(void)
{
	LOG_FOR_EXEMPLIFICATION_TEARDOWN_TEST;
	TEST_DONE;
}

_TEST test_1(void)
{
	LOG_FOR_EXEMPLIFICATION_TEST_CASE_1;
	TEST_DONE;
}

_TEST test_2(void)
{
	LOG_FOR_EXEMPLIFICATION_TEST_CASE_2;
	TEST_DONE;
}

_TEST test_3(void)
{
	LOG_FOR_EXEMPLIFICATION_TEST_CASE_3;
	TEST_DONE;
}

/*
B+R UnitTest: This is generated code.
Do not edit! Do not move!
Description: UnitTest Testprogramm infrastructure (TestSet).
LastUpdated: 2015-04-14 12:03:48Z
By B+R UnitTest Helper Version: 2.0.0.0
*/
UNITTEST_FIXTURES(fixtures)
{
	new_TestFixture("test_1", test_1),
	new_TestFixture("test_2", test_2),
	new_TestFixture("test_3", test_3),
};

UNITTEST_CALLER_COMPLETE_EXPLICIT(test_SetTestCases_TestSetup_TestTeardown, "test_SetTestCases_TestSetup_TestTeardown", setupTest, teardownTest, fixtures, 0, 0, cyclicSetCaller);
```

#### test_SetComplete.c
```c
/********************************************************************
* COPYRIGHT -- Bernecker + Rainer
********************************************************************
* Program: SPL_Behavior
* Author: B+R
********************************************************************
* This test set shows the sequence of calls within a test set
* Add some busy conditions or test cases to see the changes.
********************************************************************/

#include <bur/plctypes.h>

#ifdef _DEFAULT_INCLUDES
#include <AsDefault.h>
#endif

#include "UnitTest.h"

#include "iHelperFunction.h"

void resetDataForTestSet_Complete()
{
	resetDataForTestSet();
}

_CYCLIC_SET(void)
{
	LOG_FOR_EXEMPLIFICATION_CYCLIC_SET;
	return;
}

_SETUP_SET(void)
{
	LOG_FOR_EXEMPLIFICATION_SETUP_SET;
	TEST_DONE;
}

_TEARDOWN_SET(void)
{
	LOG_FOR_EXEMPLIFICATION_TEARDOWN_SET;
	TEST_DONE;
}

_SETUP_TEST(void)
{
	LOG_FOR_EXEMPLIFICATION_SETUP_TEST;
	TEST_DONE;
}

_TEARDOWN_TEST(void)
{
	LOG_FOR_EXEMPLIFICATION_TEARDOWN_TEST;
	TEST_DONE;
}

_TEST test_1(void)
{
	LOG_FOR_EXEMPLIFICATION_TEST_CASE_1;
	TEST_DONE;
}

_TEST test_2(void)
{
	LOG_FOR_EXEMPLIFICATION_TEST_CASE_2;
	TEST_DONE;
}

_TEST test_3(void)
{
	LOG_FOR_EXEMPLIFICATION_TEST_CASE_3;
	TEST_DONE;
}

/*
B+R UnitTest: This is generated code.
Do not edit! Do not move!
Description: UnitTest Testprogramm infrastructure (TestSet).
LastUpdated: 2015-04-14 12:03:48Z
By B+R UnitTest Helper Version: 2.0.0.0
*/
UNITTEST_FIXTURES(fixtures)
{
	new_TestFixture("test_1", test_1),
	new_TestFixture("test_2", test_2),
	new_TestFixture("test_3", test_3),
};

UNITTEST_CALLER_COMPLETE_EXPLICIT(test_SetComplete, "test_SetComplete", setupTest, teardownTest, fixtures, setupSet, teardownSet, cyclicSetCaller);
```

#### TestBusy_AsyncronousVariables.var - Variables used in sub package "TestBusy_Asyncronous"
```iecst
(********************************************************************
 * COPYRIGHT -- Bernecker + Rainer
 ********************************************************************
 * Program: SPL_Behavior
 * Author: B+R
 ********************************************************************
 * Local variables of program SPL_Behavior
 * For test sets in package TestBusy_Asyncronous
 ********************************************************************)
VAR
	GetMimeTypeResult : STRING[80] := '';
	webserverStatus : CfgGetWebServerStatus := (0);
	webserverGetMimeType : CfgGetWebMimeType := (0);
	webserverSetMimeType : CfgSetWebMimeType := (0);
END_VAR
```

#### Package Logical/TS_UnitTest/Samples/Framework_Features/SPL_Behavior/TestBusy_Asyncronous - Testing FBs / testing with a busy condition

#### TestBusy_Asyncronous.c
```c
/********************************************************************
* COPYRIGHT -- Bernecker + Rainer
********************************************************************
* Program: SPL_Behavior
* Author: B+R
********************************************************************
* This test set shows the option to call a function
*       (test case, setup or teardown) until "done".
* This is usable for example for testing asynchronous FUBs.
********************************************************************/

#include <bur/plctypes.h>

#ifdef _DEFAULT_INCLUDES
#include <AsDefault.h>
#endif

#include "AsArCfg.h"

#include "UnitTest.h"

/* _SETUP_TEST() is called before each test case of this test set */
_SETUP_TEST(void)
{
	/* Call */
	webserverStatus.enable = 0;
	CfgGetWebServerStatus(&webserverStatus);

	webserverSetMimeType.enable = 0;
	CfgSetWebMimeType(&webserverSetMimeType);

	webserverGetMimeType.enable = 0;
	CfgGetWebMimeType(&webserverGetMimeType);

	/* Done */
	TEST_DONE;
}

/* _TEARDOWN_SET() is called at end of this test set */
_TEARDOWN_SET(void)
{
	/* Call */
	webserverStatus.enable = 0;
	CfgGetWebServerStatus(&webserverStatus);

	webserverSetMimeType.enable = 0;
	CfgSetWebMimeType(&webserverSetMimeType);

	webserverGetMimeType.enable = 0;
	CfgGetWebMimeType(&webserverGetMimeType);

	/* Done */
	TEST_DONE;
}

/* Sample test case tests async. FB CfgGetWebServerStatus() */
_TEST test_AsyncFub(void)
{
	/* Call */
	webserverStatus.enable = 1;
	CfgGetWebServerStatus(&webserverStatus);

	/* Wait  */
	TEST_BUSY_CONDITION(ERR_FUB_BUSY == webserverStatus.status );

	/* Test */
	TEST_ASSERT_EQUAL_INT( ERR_OK, webserverStatus.status  );
	TEST_ASSERT_EQUAL_INT(cfgWEB_MODE_ENABLED,  webserverStatus.mode);

	/* Done */
	TEST_DONE;
}

/* Sample test case tests async. FB CfgGetWebMimeType() */
_TEST test_getMimeType(void)
{
	/* Call */
	webserverGetMimeType.enable = 1;
	webserverGetMimeType.pFileExtension =  (UDINT) "*.txt";
	webserverGetMimeType.pMimeType = (UDINT)GetMimeTypeResult;
	webserverGetMimeType.len = sizeof(GetMimeTypeResult) - 1;
	CfgGetWebMimeType(&webserverGetMimeType);

	/* Wait  */
	TEST_BUSY_CONDITION_MSG(ERR_FUB_BUSY == webserverGetMimeType.status,  "Fub is busy");

	/* Test */
	TEST_ASSERT_EQUAL_INT( ERR_OK, webserverGetMimeType.status  );
	TEST_ASSERT_EQUAL_STRING("text/plain", GetMimeTypeResult   );

	/* Done */
	TEST_DONE;
}

/*
B+R UnitTest: This is generated code.
Do not edit! Do not move!
Description: UnitTest Testprogramm infrastructure (TestSet).
LastUpdated: 2015-04-14 12:03:48Z
By B+R UnitTest Helper Version: 2.0.0.0
*/
UNITTEST_FIXTURES(fixtures)
{
	new_TestFixture("test_AsyncFub", test_AsyncFub),
	new_TestFixture("test_getMimeType", test_getMimeType),
};

UNITTEST_CALLER_COMPLETE_EXPLICIT(TestBusy_Asyncronous, "TestBusy_Asyncronous", setupTest, 0, fixtures, 0, teardownSet, 0);
```

#### TestBusy_Asyncronous_with_CyclicSet.c - This test set adds additional information to the test report (for illustration only)
```c
/********************************************************************
* COPYRIGHT -- Bernecker + Rainer
********************************************************************
* Program: SPL_Behavior
* Author: B+R
********************************************************************
* This test set shows the option to call a function
*       (test case, setup or teardown) until "done".
* This is usable for example for testing asynchronous FUBs.
********************************************************************/

#include <bur/plctypes.h>

#ifdef _DEFAULT_INCLUDES
#include <AsDefault.h>
#endif

#include "UnitTest.h"

#include "iHelperFunction.h"

/*_CYCLIC_SET() is called in each cycle as long this Test Set is the active test set*/
_CYCLIC_SET(void)
{
	LOG_FOR_EXEMPLIFICATION_CYCLIC_SET;
	CfgGetWebServerStatus(&webserverStatus);
	CfgSetWebMimeType(&webserverSetMimeType);
	CfgGetWebMimeType(&webserverGetMimeType);

}

/* _SETUP_SET() is called at the beginning of this test set */
_SETUP_SET(void)
{
	resetDataForTestSet();

	LOG_FOR_EXEMPLIFICATION_SETUP_SET;

	/*Disable FB at beginning of this test set*/
	webserverStatus.enable = 0;
	webserverSetMimeType.enable = 0;
	webserverGetMimeType.enable = 0;

	TEST_DONE;
}

/* _SETUP_TEST() is called before each test case of this test set */
_SETUP_TEST(void)
{
	LOG_FOR_EXEMPLIFICATION_SETUP_TEST;

	/*Disable FB at beginning of this test set*/
	webserverStatus.enable = 0;
	webserverSetMimeType.enable = 0;
	webserverGetMimeType.enable = 0;

	TEST_DONE;
}

/* _TEARDOWN_SET() is called at end of this test set */
_TEARDOWN_SET(void)
{
	LOG_FOR_EXEMPLIFICATION_TEARDOWN_SET;
	/*Disable FB after each test case*/
	webserverStatus.enable = 0;
	webserverSetMimeType.enable = 0;
	webserverGetMimeType.enable = 0;

	/* Done */
	TEST_DONE;
}

/* Sample test case tests async. FB CfgGetWebServerStatus() */
_TEST test_AsyncFub(void)
{
	LOG_FOR_EXEMPLIFICATION_TEST_CASE_1;

	/*Silent  wait  as FB is still busy*/
	TEST_BUSY_CONDITION(ERR_FUB_BUSY == webserverStatus.status  );

	webserverStatus.enable = 1;

	/*Silent  wait  as FB is not yet enabled*/
	TEST_BUSY_CONDITION( ERR_FUB_ENABLE_FALSE == webserverStatus.status );

	/* Test */
	TEST_ASSERT_EQUAL_INT( ERR_OK, webserverStatus.status  );
	TEST_ASSERT_EQUAL_INT(cfgWEB_MODE_ENABLED,  webserverStatus.mode);

	/* Done */
	TEST_DONE;
}

/* Sample test case tests async. FB CfgGetWebMimeType() */
_TEST test_getMimeType(void)
{
	LOG_FOR_EXEMPLIFICATION_TEST_CASE_3;

	TEST_BUSY_CONDITION_MSG(ERR_FUB_BUSY == webserverGetMimeType.status,  "Fub is busy");

	webserverGetMimeType.enable = 1;
	webserverGetMimeType.pFileExtension =  (UDINT) "*.txt";
	webserverGetMimeType.pMimeType = (UDINT)GetMimeTypeResult;
	webserverGetMimeType.len = sizeof(GetMimeTypeResult) - 1;

	/* Wait  */
	TEST_BUSY_CONDITION_MSG(ERR_FUB_ENABLE_FALSE == webserverGetMimeType.status,  "Fub is not enabled");

	/* Test */
	TEST_ASSERT_EQUAL_INT( ERR_OK, webserverGetMimeType.status  );
	TEST_ASSERT_EQUAL_STRING("text/plain", GetMimeTypeResult   );

	/* Done */
	TEST_DONE;
}

/*
B+R UnitTest: This is generated code.
Do not edit! Do not move!
Description: UnitTest Testprogramm infrastructure (TestSet).
LastUpdated: 2015-04-14 12:03:48Z
By B+R UnitTest Helper Version: 2.0.0.0
*/
UNITTEST_FIXTURES(fixtures)
{
	new_TestFixture("test_AsyncFub", test_AsyncFub),
	new_TestFixture("test_getMimeType", test_getMimeType),
};

UNITTEST_CALLER_COMPLETE_EXPLICIT(TestBusy_Asyncronous_with_CyclicSet, "TestBusy_Asyncronous_with_CyclicSet", setupTest, 0, fixtures, setupSet, teardownSet, cyclicSetCaller);
```

### Package Logical/TS_UnitTest/Templates/HelperTool_Supported - Easy mode: focus on writing tests

### Steps.txt
```
Precondition: UnitTest Libraries are added to current active configuration
	(See AS help:  Solutions - Technology solutions - Unit test - Getting started - Adjusting the target configuration)

1. 	Copy template program
2. 	Rename the copy of the template program
3. 	Rename TestSuite.Name
4. 	Copy test set template

5. 	Implement test case
6. 	Copy batch file "Update_TestPrograms_in_current_location.bat" if it is not already in destination package
7. 	Double click batch file

8. 	Add test program to active software configuration
9.	Compile & transfer
10. Refresh test list in the test view
11. Run test
```

### Program Logical/TS_UnitTest/Templates/HelperTool_Supported/utTemplate_automated (ANSIC) - Empty template for use with helper tool

#### variables.var - Name the suite and add PVs for the program
```iecst
(********************************************************************
 * COPYRIGHT --
 ********************************************************************
 * Program: utTemplate_automated
 * File: variables.var
 * Author: -
 * Created: -
 ********************************************************************
 * Local variables of program utTemplate_automated
 ********************************************************************)
(*Describe the test*)
VAR
	Testsuite : UtMgrTestSuite := (Name:='automatedTemplate_ToBeRenamed',Description:='(Optional field)Template for use with helper tool. Reference or add this program in the package "TS_UnitTest_UpdateTestPrograms"',Type:=utMgrTEST_TYPE_C,MetaInformation:='(Optional field):To be filled');
END_VAR
(*Variables used in the tests*)
```

#### testSuite.c
```c
/********************************************************************
 * COPYRIGHT --
 ********************************************************************
 * Program: -
 * Author:
 * Created:
 ********************************************************************
 * Test registration and handshake
 ********************************************************************/

#include <bur/plctypes.h>

#ifdef _DEFAULT_INCLUDES
#include <AsDefault.h>
#endif

#include "UnitTest.h"

void _INIT initTestSuite(void)
{
	utInit(&Testsuite);
}

void _CYCLIC cyclicWithTest(void)
{
	utCyclic(&Testsuite);
}

void _EXIT exitTestSuite(void)
{
	utExit(&Testsuite);
}
```

#### autoGeneratedFile.c - Auto generated code - list of all test sets in the program
```c
/* This content will be auto updated by the helper tool */

#include "UnitTest.h"

UNITTEST_TESTSET_FIXTURES (utTestSets)
{
	{
		0
	}
};
UNTITTEST_TESTSET_HANDLER();
```

### Package Logical/TS_UnitTest/Templates/HelperTool_Supported/TestSet_Templates - Multiple variants of valid test sets

### Set_Complete.c
```c
/********************************************************************
 * COPYRIGHT --
 ********************************************************************
 * Program: -
 * Author:
 * Created:
 ********************************************************************
 * Tests for ...
 ********************************************************************/

#include <bur/plctypes.h>

#ifdef _DEFAULT_INCLUDES
#include <AsDefault.h>
#endif

#include "UnitTest.h"

_CYCLIC_SET()
{

	/* TODO:  add code running cyclically while test set is active here */
	return;
}

_SETUP_SET(void)
{
	/* TODO:  add code running before test set here */
	TEST_DONE;
}

_TEARDOWN_SET(void)
{
	/* TODO:  add code running after test set here */
	TEST_DONE;
}

_SETUP_TEST(void)
{
	/* TODO:  add code running before test case here */
	TEST_DONE;
}

_TEARDOWN_TEST(void)
{
	/* TODO:  add code running after test case here */
	TEST_DONE;
}

_TEST testcase1(void)
{

	/* TODO:  add assertions here */

	/* test is done */
	TEST_DONE;
}
```

### Set_SetupTeardown.c
```c
/********************************************************************
 * COPYRIGHT --
 ********************************************************************
 * Program: -
 * Author:
 * Created:
 ********************************************************************
 * Tests for ...
 ********************************************************************/

#include <bur/plctypes.h>

#ifdef _DEFAULT_INCLUDES
#include <AsDefault.h>
#endif

#include "UnitTest.h"

_SETUP_SET(void)
{
	/* TODO:  add code running before test set here */
	TEST_DONE;
}

_TEARDOWN_SET(void)
{
	/* TODO:  add code running after test set here */
	TEST_DONE;
}

_SETUP_TEST(void)
{
	/* TODO:  add code running before test case here */
	TEST_DONE;
}

_TEARDOWN_TEST(void)
{
	/* TODO:  add code running after test case here */
	TEST_DONE;
}

_TEST testcase1(void)
{

	/* TODO:  add assertions here */

	/* test is done */
	TEST_DONE;
}
```

### Set_Testcases.c
```c
/********************************************************************
 * COPYRIGHT --
 ********************************************************************
 * Program: -
 * Author:
 * Created:
 ********************************************************************
 * Tests for ...
 ********************************************************************/

#include <bur/plctypes.h>

#ifdef _DEFAULT_INCLUDES
#include <AsDefault.h>
#endif

#include "UnitTest.h"

_TEST testcase1(void)
{

	/* TODO:  add assertions here */

	/* test is done */
	TEST_DONE;
}
```

- Update_TestPrograms_in_current_location.bat - Updates test programs within the current package (not shown)

### Package Logical/TS_UnitTest/Templates/NoToolSupport - Advanced mode: more control over fixtures

### Program Logical/TS_UnitTest/Templates/NoToolSupport/utTemplate_manual (ANSIC) - Empty Template without support of helper tool

#### variables.var - Name the suite and add PVs for the program
```iecst
(********************************************************************
 * COPYRIGHT --
 ********************************************************************
 * Program: utTemplate_manual
 * File: variables.var
 * Author: -
 * Created: -
 ********************************************************************
 * Local variables of program utTemplate_manual
 ********************************************************************)
(*Describe the test*)
VAR
	Testsuite : UtMgrTestSuite := (Name:='manualTemplate_ToBeRenamed',Description:='(Optional field): Template to manually update the infrastructure (fixtures of test cases and sets)',Type:=utMgrTEST_TYPE_C,MetaInformation:='(Optional field):To be filled');
END_VAR
(*Variables used in the tests*)
```

#### testSuite.c - No changes needed
```c
/********************************************************************
 * COPYRIGHT --
 ********************************************************************
 * Program: -
 * Author:
 * Created:
 ********************************************************************
 * Test registration and handshake
 ********************************************************************/

#include <bur/plctypes.h>

#ifdef _DEFAULT_INCLUDES
#include <AsDefault.h>
#endif

#include "UnitTest.h"

void _INIT initTestSuite(void)
{
	utInit(&Testsuite);
}

void _CYCLIC cyclicWithTest(void)
{
	utCyclic(&Testsuite);
}

void _EXIT exitTestSuite(void)
{
	utExit(&Testsuite);
}
```

#### FixtureOfTestSets.c - List of test sets, all test sets of the program have to be added here
```c
/********************************************************************
 * COPYRIGHT --
 ********************************************************************
 * Program: -
 * Author:
 * Created:
 ********************************************************************
 * Test Set Fixture
 ********************************************************************/

#include "UnitTest.h"

/* TODO: Add your sets here

UNITTEST_TESTSET_DECLARATION testSet1;
UNITTEST_TESTSET_DECLARATION testSet2;
*/

/* List of all test sets of the test programm
they will be executed in the given order*/
UNITTEST_TESTSET_FIXTURES (utTestSets)
{
#warning TODO: Add your sets here
	/* TODO: Add your sets here
	new_TestSet(testSet1),
	new_TestSet(testSet2)*/
	{
		0
	} /* Place holder for test sets, can be removed */
};

/*Handler of test set list */
UNTITTEST_TESTSET_HANDLER();
```

### Package Logical/TS_UnitTest/Templates/NoToolSupport/TestSet_Templates - Multiple variants of valid test sets

### Set_Testcases.c
```c
/********************************************************************
 * COPYRIGHT --
 ********************************************************************
 * Program: -
 * Author:
 * Created:
 ********************************************************************
 * Tests for ...
 ********************************************************************/

#include <bur/plctypes.h>

#ifdef _DEFAULT_INCLUDES
#include <AsDefault.h>
#endif

#include "UnitTest.h"

/* a test case*/
_TEST testcase1(void)
{

	/* TODO: add assertions here */

	/* test is done */
	TEST_DONE;
}

/* a test case*/
_TEST testcase2(void)
{
	/* TODO: add assertions here */

	/* test is done */
	TEST_DONE;
}

#warning TODO: Add your test cases here
/*TODO: Add your test cases here */
UNITTEST_FIXTURES(fixtures)
{
	new_TestFixture("testcase1",testcase1),
	                new_TestFixture("testcase2",testcase2),
};

#warning TODO: rename testset (Param 1 and 2)
UNITTEST_CALLER_TEST(testSet_testcases, "testSet_testcases",fixtures);
```

### Set_SetupTeardown.c
```c
/********************************************************************
 * COPYRIGHT --
 ********************************************************************
 * Program: -
 * Author:
 * Created:
 ********************************************************************
 * Tests for ...
 ********************************************************************/

#include <bur/plctypes.h>

#ifdef _DEFAULT_INCLUDES
#include <AsDefault.h>
#endif

#include "UnitTest.h"

/* called before first test case of test set*/
_SETUP_SET(void)
{
	/* TODO:  add code running before test set here */
	TEST_DONE;
}

/* called after last test case of test set */
_TEARDOWN_SET(void)
{
	/* TODO:  add code running after test set here */
	TEST_DONE;
}

/* called before a test case first called */
_SETUP_TEST(void)
{
	/* TODO:  add code running before test case here */
	TEST_DONE;
}

/* called after a test case is done*/
_TEARDOWN_TEST(void)
{
	/* TODO:  add code running after test case here */
	TEST_DONE;
}

/* ---------------------------*/

/* a test case*/
_TEST testcase1(void)
{

	/* TODO:  add assertions here */

	/* test is done */
	TEST_DONE;
}

/* a test case*/
_TEST testcase2(void)
{
	/* TODO:  add assertions here */

	/* test is done */
	TEST_DONE;
}

#warning TODO: Add your test cases here
/*TODO: Add your test cases here */
UNITTEST_FIXTURES(fixtures)
{
	new_TestFixture("testcase1",testcase1),
	                new_TestFixture("testcase2",testcase2),
};

#warning TODO: rename testset (Param 1 and 2)
UNITTEST_CALLER_SET(testSetupTeardown, "testSetupTeardown",fixtures);
```

### Set_Complete.c
```c
/********************************************************************
 * COPYRIGHT --
 ********************************************************************
 * Program: -
 * Author:
 * Created:
 ********************************************************************
 * Tests for ...
 ********************************************************************/

#include <bur/plctypes.h>

#ifdef _DEFAULT_INCLUDES
#include <AsDefault.h>
#endif

#include "UnitTest.h"

/* called when test set is active. */
_CYCLIC_SET()
{

	/* TODO:  add code running cyclically while test set is active here */
	return;
}

/* called before first test case of test set*/
_SETUP_SET(void)
{
	/* TODO:  add code running before test set here */
	TEST_DONE;
}

/* called after last test case of test set */
_TEARDOWN_SET(void)
{
	/* TODO:  add code running after test set here */
	TEST_DONE;
}

/* called before a test case first called */
_SETUP_TEST(void)
{
	/* TODO:  add code running before test case here */
	TEST_DONE;
}

/* called after a test case is done*/
_TEARDOWN_TEST(void)
{
	/* TODO:  add code running after test case here */
	TEST_DONE;
}
/* ---------------------------*/

/* a test case*/
_TEST testcase1(void)
{

	/* TODO:  add assertions here */

	/* test is done */
	TEST_DONE;
}

/* a test case*/
_TEST testcase2(void)
{
	/* TODO:  add assertions here */

	/* test is done */
	TEST_DONE;
}

#warning TODO: Add your test cases here
/*TODO: Add your test cases here */
UNITTEST_FIXTURES(fixtures)
{
	new_TestFixture("testcase1",testcase1),
	                new_TestFixture("testcase2",testcase2),
};

#warning TODO: rename testset (Param 1 and 2)
UNITTEST_CALLER_COMPLETE(testSetComplete, "testSetComplete",fixtures);
```

Listed in the project but not available here: Logical/Global.typ, Logical/TS_UnitTest/Samples/Framework_Extension_With_Custom_Asserts/LibAssert1/LibAssert1.h, Logical/TS_UnitTest/Samples/Framework_Extension_With_Custom_Asserts/LibAssert1/LibAssert1_ThresholdAssert.h, Logical/TS_UnitTest/Samples/Framework_Extension_With_Custom_Asserts/LibAssert1/LibAssert1_ThresholdAssert.c, Logical/TS_UnitTest/Samples/Framework_Extension_With_Custom_Asserts/LibAssert1/LibAssert1_REAL_ArrayAsserts.h, Logical/TS_UnitTest/Samples/Framework_Extension_With_Custom_Asserts/LibAssert1/LibAssert1_REAL_ArrayAsserts.c
